Fanuc KAREL source: abs.kl

PROGRAM mth_abs
%NOBUSYLAMP
%NOLOCKGROUP
%COMMENT = 'absolute value'

VAR
	  reg_no : INTEGER
    val : REAL

%include tpe.klh
%include registers.klh


BEGIN
  val = tpe__get_real_arg(1)
  reg_no = tpe__get_int_arg(2)

  registers__set_real(reg_no, ABS(val))
END mth_abs
